FUNCTION alg_a_transfer2droppos : BOOL
VAR_INPUT
	state: STATE;
END_VAR

alg_a_transfer2droppos := state.dvar_M_vacuum_a_transfer2droppos;

END_FUNCTION

(* stored: Version 1.1.0.1, ProductVersion 3.1.4022.18
   POU alg_a_transfer2droppos: Id {4ac6413b-47ff-41e2-a16c-d76a11a28c98}, SpecialFunc None *)
